TYPE ST_Camera_OUT :
STRUCT
	nPLCType						:UINT;
	nControlStatus					:UINT;
END_STRUCT
END_TYPE

(* stored: Version 1.1.0.1, ProductVersion 3.1.4024.10
   DUT ST_Camera_OUT: Id {e90c5630-ad47-46c4-a1ee-7f1cc572759c} *)
